(* CODESYS project CODESYS SIMULATION 1.project

Project tree, tasks and I/O mapping:
  Device : CODESYS Control Win V3, 3S - Smart Software Solutions GmbH, order no. 305021, version 3.5.9.10
    application Application
      libraries: Standard, * (System)
      task MainTask (cyclic, interval t#20ms, priority 1) calls PLC_PRG
      task VISU_TASK (cyclic, interval 100 ms, priority 31) calls VisuElems.Visu_Prg
      program PLC_PRG [ST]
      Symbols
      global variables GVL
      visualisation Visualization
  libraries: VisuSymbols, 3.5.8.0 (System)
  5ce3da45-db07-42e7-a21c-a00fff4ed8f6|C:\Users\J.A.F.M\Downloads\ICONO BRAZO VENTOSA.png
  text list GlobalTextList
  image pool ImagePool
*)

// Device/Application/GVL
VAR_GLOBAL
	entradas_plc1: BYTE;
	entradas_plc2: BYTE;
	entradas_plc3: BYTE;
	salidas_plc1: BYTE;
	salidas_plc2: BYTE;
	salidas_plc3: BYTE;
END_VAR

// Device/Application/PLC_PRG
PROGRAM PLC_PRG
VAR
	LED_START: BOOL;
	LED_STOP: BOOL;
	LED_EMERGENCIA: BOOL;
END_VAR

//Logica de programación//

//Entradas Codesys//

//START = entradas_plc2.5; //
//STOP = entradas_plc2.6; //
//EMERGENCIA = entradas_plc2.7; //

//CAJAS ENTRADA//
//CAJA 1 = entradas_plc1.2;
//CAJA 2 = entradas_plc1.3;
//CAJA 3 = entradas_plc1.4;
//CAJA 4 = entradas_plc1.5;
//CAJA 5 = entradas_plc1.6;
//CAJA 6 = entradas_plc1.7;
//CAJA 7 = entradas_plc2.0;
//CAJA 8 = entradas_plc2.1;

//Salidas Fluidsim//
//salidas_plc2.5;//
//salidas_plc2.6;//
//salidas_plc2.7;//

//STAR-STOP-EMERGENCIA//

// SALIDA STOP (activa si STOP o EMERGENCIA)
IF NOT entradas_plc2.6 OR NOT entradas_plc2.7 THEN
    salidas_plc2.6 := TRUE;
ELSE
    salidas_plc2.6 := FALSE;
END_IF

// SALIDA EMERGENCIA
IF NOT entradas_plc2.7 THEN
    salidas_plc2.7 := TRUE;
ELSE
    salidas_plc2.7 := FALSE;
END_IF

// MARCHA ENCLAVADA
IF NOT entradas_plc2.6 OR NOT entradas_plc2.7 THEN
    salidas_plc2.5 := FALSE;
ELSIF entradas_plc2.5 THEN
    salidas_plc2.5 := TRUE;
END_IF

//LEDS START-STOP-EMERGENCIA//
//LED START//
IF salidas_plc2.5:= TRUE THEN LED_START:= TRUE;
	ELSE LED_START:= FALSE; 
END_IF

//LED STOP//
IF salidas_plc2.6:= FALSE THEN LED_STOP:= TRUE;
	ELSE LED_STOP:= FALSE; 
END_IF

//LED EMERGENCIA//
IF salidas_plc2.7:= FALSE THEN LED_EMERGENCIA:= TRUE;
	ELSE LED_EMERGENCIA:= FALSE; 
END_IF



// LED CAJA 1
IF entradas_plc1.2 THEN 
    salidas_plc1.2:=TRUE;
ELSE 
    salidas_plc1.2:=FALSE;
END_IF

// LED CAJA 2
IF entradas_plc1.3 THEN 
    salidas_plc1.3:=TRUE;
ELSE 
    salidas_plc1.3:=FALSE;
END_IF

// LED CAJA 3
IF entradas_plc1.4 THEN 
    salidas_plc1.4:=TRUE;
ELSE 
    salidas_plc1.4:=FALSE;
END_IF

// LED CAJA 4
IF entradas_plc1.5 THEN 
    salidas_plc1.5:=TRUE;
ELSE 
    salidas_plc1.5:=FALSE;
END_IF

// LED CAJA 5
IF entradas_plc1.6 THEN 
    salidas_plc1.6:=TRUE;
ELSE 
    salidas_plc1.6:=FALSE;
END_IF

// LED CAJA 6
IF entradas_plc1.7 THEN 
    salidas_plc1.7:=TRUE;
ELSE 
    salidas_plc1.7:=FALSE;
END_IF

// LED CAJA 7
IF entradas_plc2.0 THEN 
    salidas_plc2.0:=TRUE;
ELSE 
    salidas_plc2.0:=FALSE;
END_IF

// LED CAJA 8
IF entradas_plc2.1 THEN 
    salidas_plc2.1:=TRUE;
ELSE 
    salidas_plc2.1:=FALSE;
END_IF
//Puertos sin uso//
salidas_plc2.7 := FALSE;

END_PROGRAM

// Device/Application/Visualization
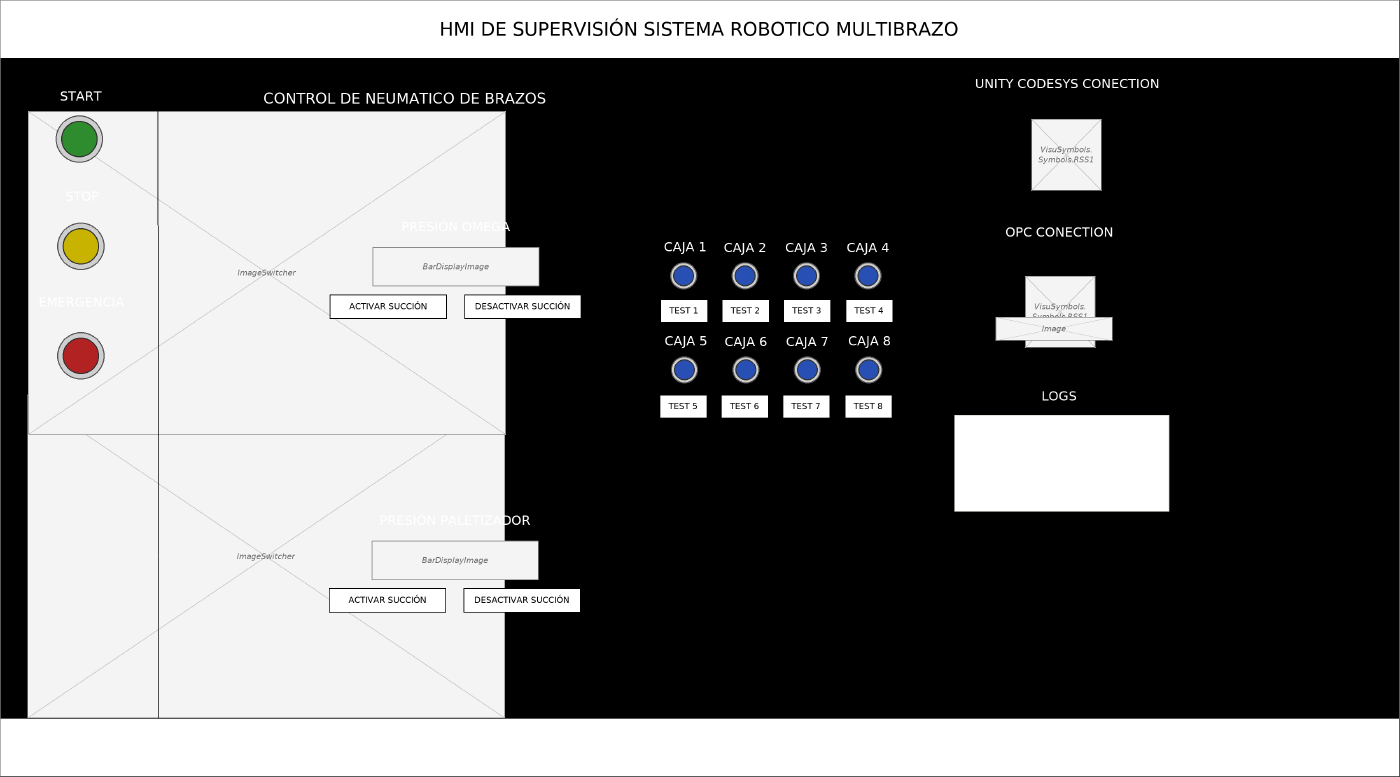
VISUALIZATION Visualization  // 1800x1000
    ImageSwitcher (35,508 614x416), image: ImagePool.0, behaviour: TOGGLE
    ImageSwitcher (36,143 614x416), image: ImagePool.0, behaviour: TOGGLE
    Label (29,109 150x30), "START"
    Rectangle (-1,0 1800x75), "HMI DE SUPERVISIÓN SISTEMA ROBOTICO MULTIBRAZO"
    Lamp1 (67,144 70x70), tooltip "START", variable: PLC_PRG.LED_START, style: Lamp-Lamp1-Green
    Lamp1 (69,282 70x70), tooltip "STOP", variable: PLC_PRG.LED_STOP, style: Lamp-Lamp1-Yellow
    Lamp1 (69,423 70x70), tooltip "EMERGENCIA", variable: PLC_PRG.LED_EMERGENCIA, style: Lamp-Lamp1-Red
    Label (31,238 150x30), "STOP"
    Label (30,374 150x30), "EMERGENCIA"
    Lamp1 (859,335 40x40), style: Lamp-Lamp1-Blue
    Lamp1 (938,335 40x40), style: Lamp-Lamp1-Blue
    Label (806,303 150x30), "CAJA 1"
    Label (883,304 150x30), "CAJA 2"
    Lamp1 (1017,335 40x40), style: Lamp-Lamp1-Blue
    Label (962,304 150x30), "CAJA 3"
    Label (1041,304 150x30), "CAJA 4"
    Lamp1 (1096,335 40x40), style: Lamp-Lamp1-Blue
    Lamp1 (860,456 40x40), style: Lamp-Lamp1-Blue
    Lamp1 (939,456 40x40), style: Lamp-Lamp1-Blue
    Label (807,424 150x30), "CAJA 5"
    Label (884,425 150x30), "CAJA 6"
    Lamp1 (1018,456 40x40), style: Lamp-Lamp1-Blue
    Label (963,425 150x30), "CAJA 7"
    Label (1043,424 150x30), "CAJA 8"
    Lamp1 (1097,456 40x40), style: Lamp-Lamp1-Blue
    Rectangle (849,385 61x30), "TEST 1"
    Rectangle (928,385 61x30), "TEST 2"
    Rectangle (1007,385 61x30), "TEST 3"
    Rectangle (1087,385 61x30), "TEST 4"
    Rectangle (848,508 61x30), "TEST 5"
    Rectangle (927,508 61x30), "TEST 6"
    Rectangle (1006,508 61x30), "TEST 7"
    Rectangle (1086,508 61x30), "TEST 8"
    BarDisplayImage (479,318 214x50), style: BarDisplayImage-Gray, scale format: %.1f, scale 0..100
    Label (478,277 216x30), "PRESIÓN OMEGA"
    Rectangle (424,379 150x31), "ACTIVAR SUCCIÓN"
    Rectangle (597,379 150x31), "DESACTIVAR SUCCIÓN"
    Label (322,112 397x30), "CONTROL DE NEUMATICO DE BRAZOS"
    Label (1254,284 216x30), "OPC CONECTION"
    Label (1231,93 283x30), "UNITY CODESYS CONECTION"
    Label (1254,495 216x30), "LOGS"
    Line (204,929) (203,77)
    Line (12,711)
    Rectangle (-1,924 1801x75)
    Image (1326,153 90x92), image: VisuSymbols.Symbols.RSS1
    Image (1318,355 90x92), image: VisuSymbols.Symbols.RSS1
    Textfield (1227,534 276x124)
    Image (1280,408 150x30)
    BarDisplayImage (478,696 214x50), style: BarDisplayImage-Gray, scale format: %.1f, scale 0..100
    Label (477,655 216x30), "PRESIÓN PALETIZADOR"
    Rectangle (423,757 150x31), "ACTIVAR SUCCIÓN"
    Rectangle (596,757 150x31), "DESACTIVAR SUCCIÓN"
END_VISUALIZATION
